TYPE PALLET :
STRUCT
	EX : BOOL:=FALSE;
	WS2 : BOOL:=FALSE;
	WS3 : BOOL:=FALSE;
	POSITION : INT:=-1;
	NEXT_PALLET : INT:=0;
	PREVIOUS_PALLET : INT:=0;
	NUMBER : INT;
END_STRUCT
END_TYPE

(* stored: Version 1.1.0.1, ProductVersion 3.1.4020.6
   DUT PALLET: Id {73f05eb7-54a7-44a4-a1b6-5b709b175cae} *)
